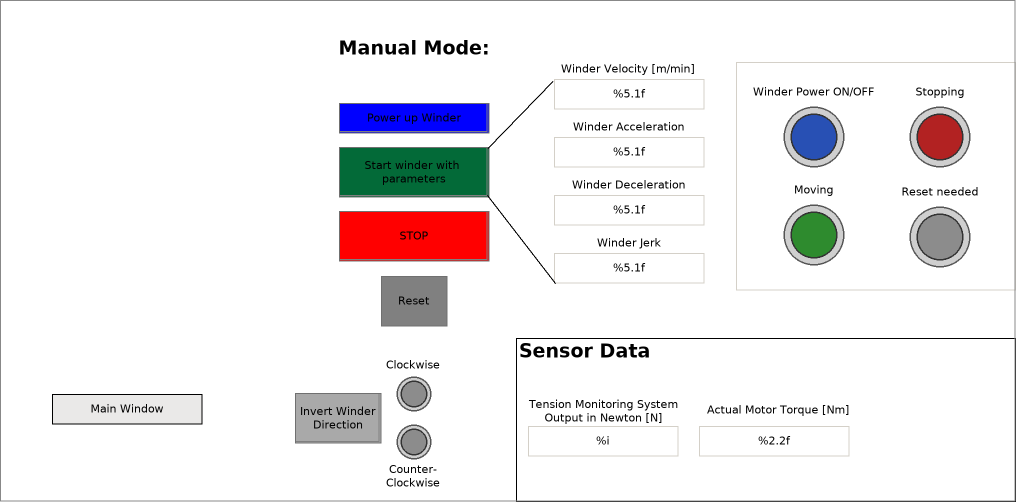
VISUALIZATION Manual_Mode  // 1016x502
    Rectangle (52,394 150x30), "Main Window"
        OnMouseClick: change screen: MainWindow
    Textfield (736,62 280x228)
    Textfield (516,338 500x164), "Sensor Data"
    Label (328,33 172x30), "Manual Mode:"
    Textfield (554,79 150x30), "%5.1f", text variable: GVL_Axis.rWinderVelocity
        OnMouseClick: write the text variable via VisuDialogs.Numpad, min 2.7, max 15
    Label (553,54 150x30), "Winder Velocity [m/min]"
    Textfield (554,137 150x30), "%5.1f", text variable: GVL_Axis.rWinderAcceleration
        OnMouseClick: write the text variable via Default
    Label (554,112 150x30), "Winder Acceleration"
    Textfield (554,253 150x30), "%5.1f", text variable: GVL_Axis.rWinderJerk
        OnMouseClick: write the text variable via Default
    Textfield (554,195 150x30), "%5.1f", text variable: GVL_Axis.rWinderDeceleration
        OnMouseClick: write the text variable via Default
    Label (554,170 150x30), "Winder Deceleration"
    Label (554,228 150x30), "Winder Jerk"
    Button (339,103 150x30), "Power up Winder", colour toggle: GVL_HMI.bButtonWinderPower
        toggle GVL_HMI.bButtonWinderPower
    Button (339,147 150x50), "Start winder with parameters", colour toggle: GVL_HMI.bButtonStartWinder
        OnMouseDown: execute { GVL_HMI.bButtonStartWinder := TRUE; }
        OnMouseUp: execute { GVL_HMI.bButtonStartWinder := FALSE; }
    Button (339,211 150x50), "STOP", colour toggle: GVL_HMI.bButtonStopWinder
        OnMouseDown: execute { GVL_HMI.bButtonStopWinder := TRUE; }
        OnMouseUp: execute { GVL_HMI.bButtonStopWinder := FALSE; }
    Button (381,276 66x50), "Reset", colour toggle: GVL_HMI.bButtonResetWinder
        OnMouseDown: execute { GVL_HMI.bButtonResetWinder := TRUE; }
        OnMouseUp: execute { GVL_HMI.bButtonResetWinder := FALSE; }
    Line (488,148) (553,81)
    Line (487,195) (555,283)
    Lamp1 (779,102 70x70), variable: GVL_Axis.bStatusPower, style: Lamp-Lamp1-Blue
    Label (739,77 150x30), "Winder Power ON/OFF"
    Lamp1 (779,200 70x70), variable: GVL_Axis.bStateCM, style: Lamp-Lamp1-Green
    Label (739,175 150x30), "Moving"
    Group (865,77 150x195)
        Lamp1 (40,25 70x70), variable: GVL_Axis.bStateStopping, style: Lamp-Lamp1-Red
        Label (0,0 150x30), "Stopping"
        Lamp1 (40,125 70x70), variable: GVL_Axis.bStateErrorStop, style: Lamp-Lamp1-Gray
        Label (0,100 150x30), "Reset needed"
    Textfield (528,426 150x30), "%i", text variable: GVL.iTensionMonitoringData
    Label (522,396 163x30), "Tension Monitoring System Output in Newton [N]"
    Button (295,393 86x50), "Invert Winder Direction", colour toggle: GVL_HMI.bButtonWinderDirection
        toggle GVL_HMI.bButtonWinderDirection
    Lamp1 (394,374 40x40), variable: GVL_HMI.bButtonWinderDirection, style: Lamp-Lamp1-Gray
    Lamp1 (394,422 40x40), variable: GVL_HMI.bButtonNotWinderDirection, style: Lamp-Lamp1-Gray
    Label (371,350 84x30), "Clockwise"
    Label (371,461 84x30), "Counter- Clockwise"
    Textfield (699,426 150x30), "%2.2f", text variable: GVL_HMI.ActTorque
    Label (697,395 163x30), "Actual Motor Torque [Nm]"
END_VISUALIZATION

(* stored: Version 1.1.0.1
   Visu Manual_Mode: Id {41c33245-a20a-4a23-a4a6-453e0222f1a8} *)
